// TwinCAT 3 PLC project PLC1
// ProgramVersion: 3.1.4024.12
// libraries:
//   Tc2_Standard, * (Beckhoff Automation GmbH)
//   Tc2_System, * (Beckhoff Automation GmbH)
//   Tc3_Module, * (Beckhoff Automation GmbH)
// project tree:
//   FBs/Base/ FB_DriveBase.TcPOU
//   FBs/Extended/ FB_DriveCAN.TcPOU, FB_DriveNc.TcPOU
//   ITFs/ I_DriveBase.TcIO
//   / PlcTask.TcTTO
//   POUs/ MAIN.TcPOU
// real-time tasks:
//   TASK PlcTask: cycle T#10ms, priority 20, ADS port 350

CONFIGURATION PLC1
    RESOURCE PLC ON TwinCAT3
        TASK PlcTask(INTERVAL := T#10ms, PRIORITY := 20);
        PROGRAM MAIN WITH PlcTask : MAIN;
    END_RESOURCE
END_CONFIGURATION

// ---- ITFs/I_DriveBase.TcIO
INTERFACE I_DriveBase

METHOD Disable : BOOL
VAR_INPUT
END_VAR
END_METHOD

METHOD Enable : BOOL
VAR_INPUT
END_VAR
END_METHOD

METHOD MoveToPosition : BOOL
VAR_INPUT
END_VAR
END_METHOD

METHOD Reset : BOOL
VAR_INPUT
END_VAR
END_METHOD

METHOD SetLimits : BOOL
VAR_INPUT
	lrMax : LREAL;
	lrMin : LREAL;
END_VAR
END_METHOD

END_INTERFACE

// ---- POUs/MAIN.TcPOU
PROGRAM MAIN
VAR
	fbDriveNc 	: FB_DriveNC;
	fbDriveCan	: FB_DriveCAN;
	iDrive		: I_DriveBase := fbDriveNc;
	
	// Drive Swap Control
	bNcDrive: BOOL;
	bCANDrive: BOOL;
END_VAR

IF bNcDrive THEN
	bNcDrive := FALSE;
	iDrive := fbDriveNc;
END_IF

IF bCANDrive THEN
	bCANDrive := FALSE;
	iDrive := fbDriveCan;
END_IF


iDrive.Enable();

END_PROGRAM

// ---- FBs/Extended/FB_DriveNc.TcPOU
FUNCTION_BLOCK FB_DriveNc EXTENDS FB_DriveBase
VAR_INPUT
END_VAR
VAR_OUTPUT
END_VAR
VAR
END_VAR

METHOD Disable : BOOL
END_METHOD

METHOD Enable : BOOL
END_METHOD

METHOD MoveToPosition : BOOL
END_METHOD

METHOD Reset : BOOL
END_METHOD

END_FUNCTION_BLOCK

// ---- FBs/Base/FB_DriveBase.TcPOU
FUNCTION_BLOCK ABSTRACT FB_DriveBase IMPLEMENTS I_DriveBase
VAR
	lrMax : LREAL;
	lrMin : LREAL;
END_VAR

METHOD ABSTRACT Disable : BOOL
END_METHOD

METHOD ABSTRACT Enable : BOOL
END_METHOD

METHOD ABSTRACT MoveToPosition : BOOL
END_METHOD

METHOD ABSTRACT Reset : BOOL
END_METHOD

METHOD SetLimits : BOOL
VAR_INPUT
	lrMax : LREAL;
	lrMin : LREAL;
END_VAR
THIS^.lrMax := lrMax;
THIS^.lrMin := lrMin;
END_METHOD

END_FUNCTION_BLOCK

// ---- FBs/Extended/FB_DriveCAN.TcPOU
FUNCTION_BLOCK FB_DriveCAN EXTENDS FB_DriveBase
VAR_INPUT
END_VAR
VAR_OUTPUT
END_VAR
VAR
END_VAR

METHOD Disable : BOOL
END_METHOD

METHOD Enable : BOOL
END_METHOD

METHOD MoveToPosition : BOOL
END_METHOD

METHOD Reset : BOOL
END_METHOD

END_FUNCTION_BLOCK
